Yaskawa INFORM job: AAA.JBI

/JOB
//NAME AAA
//POS
///NPOS 2,0,0,0,0,0
C00000=5934,51781,-4433,23164,-46703,-28637
C00001=8424,52420,-3720,23544,-47417,-29518
//INST
///DATE 2023/02/08 10:57
///ATTR SC,RW
///GROUP1 RB1
NOP
MOVL C00000 V=10.0
MOVL C00001 V=10.0
END
